// TwinCAT 3 PLC project ProyMain
// ProgramVersion: 3.1.4024.0
// libraries:
//   CmpBitmapPool, * (System)
//   Tc2_Standard, * (Beckhoff Automation GmbH)
//   Tc2_System, * (Beckhoff Automation GmbH)
//   Tc3_Module, * (Beckhoff Automation GmbH)
//   VisuDialogs, * (System)
// project tree:
//   DUTs/ E_GEMMA.TcDUT
//   / GlobalTextList.TcGTLO, PlcTask.TcTTO, Visualization Manager.TcVMO (not stored)
//   POUs/Estacion/ FB_Coordinador_SFC.TcPOU, FB_Director.TcPOU, FB_Estacion.TcPOU
//   POUs/ MAIN.TcPOU
//   POUs/Reloj/ FB_Clock.TcPOU
//   POUs/Tareas/ FB_AlimentadorVerificadorDesplazador_SFC.TcPOU, FB_CheckMaterial_SFC.TcPOU, FB_Descargador_SFC.TcPOU, FB_EstacionFinalizar_SFC.TcPOU, FB_EstacionPreparar_SFC.TcPOU, FB_Rechazador_SFC.TcPOU, FB_ResetDescargador_SFC.TcPOU, FB_SituarPale_SFC.TcPOU, FB_TransferirPale_SFC.TcPOU
//   VISUs/ ImagePool.TcIPO (not stored), Visualization.TcVIS
// real-time tasks:
//   TASK PlcTask: cycle T#10ms, priority 20, ADS port 350
// I/O:
//   DEVICE Device 1 (EtherCAT), AmsNetId 192.168.74.1.2.1
//     Term 1 (EK1200) [EK1200-5000 EtherCAT Power supply (2A E-Bus)]
//       Term 2 (EL1008) [EL1008 8Ch. Dig. Input 24V, 3ms]
//       Term 3 (EL1008) [EL1008 8Ch. Dig. Input 24V, 3ms]
//       Term 4 (EL2008) [EL2008 8Ch. Dig. Output 24V, 0.5A]
//       Term 5 (EL2008) [EL2008 8Ch. Dig. Output 24V, 0.5A]
//       Term 6 (EL1008) [EL1008 8Ch. Dig. Input 24V, 3ms]
//       Term 7 (EL1008) [EL1008 8Ch. Dig. Input 24V, 3ms]
//       Term 8 (EL2008) [EL2008 8Ch. Dig. Output 24V, 0.5A]
//       Term 9 (EL2008) [EL2008 8Ch. Dig. Output 24V, 0.5A]
//       Term 10 (EL9011) [EL9011 End Terminal]
//   DEVICE Device 2 (EtherCAT Automation Protocol), AmsNetId 192.168.74.1.3.1
//   DEVICE Device 3 (NOV-DP-RAM)
// variable links:
//   ProyMain/ProyMain Instance <-> Device 1 (EtherCAT)/Term 1 (EK1200)/Term 2 (EL1008)
//     PlcTask Inputs/MAIN.Estacion.Codigo_pale_bit_0 <-> Channel 7/Codigo de palé bit 0
//     PlcTask Inputs/MAIN.Estacion.Codigo_pale_bit_1 <-> Channel 8/Codigo de palé bit 1
//     PlcTask Inputs/MAIN.Estacion.EstacionConectada <-> Channel 5/Parte operativa conectada (armada)
//     PlcTask Inputs/MAIN.Estacion.Presencia_pale <-> Channel 6/presencia de palé
//     PlcTask Inputs/MAIN.Estacion.Pulsador_marcha <-> Channel 3/Pulsador de marcha
//     PlcTask Inputs/MAIN.Estacion.Pulsador_parada_NC <-> Channel 4/Pulsador de parada [NC]
//     PlcTask Inputs/MAIN.Estacion.Pulsador_parada_emergencia <-> Channel 1/Pulsador de parada de emergencia
//     PlcTask Inputs/MAIN.Estacion.Selector_modo_manual <-> Channel 2/Selector de modo manual
//   ProyMain/ProyMain Instance <-> Device 1 (EtherCAT)/Term 1 (EK1200)/Term 3 (EL1008)
//     PlcTask Inputs/MAIN.Estacion.Codigo_pale_bit_2 <-> Channel 1/Código de palé bit 2
//     PlcTask Inputs/MAIN.Estacion.Detector_presion <-> Channel 2/Detector de presión
//   ProyMain/ProyMain Instance <-> Device 1 (EtherCAT)/Term 1 (EK1200)/Term 4 (EL2008)
//     PlcTask Outputs/MAIN.Estacion.Activa_marcha_motor_cinta <-> Channel 5/Activa la marcha el motor de la cinta
//     PlcTask Outputs/MAIN.Estacion.Desconecta_parte_operativa <-> Channel 1/Desconecta parte operativa (desarma)
//     PlcTask Outputs/MAIN.Estacion.Invierte_marcha_motor_cinta <-> Channel 6/Invierte la marcha del motor de la cinta
//     PlcTask Outputs/MAIN.Estacion.Lampara_falta_material <-> Channel 4/Lámpara de falta material
//     PlcTask Outputs/MAIN.Estacion.Lampara_marcha <-> Channel 3/Lámpara de marcha
//     PlcTask Outputs/MAIN.Estacion.Retenedor_pale_baja <-> Channel 7/Cilindro del retenedor de palés baja
//     PlcTask Outputs/MAIN.Estacion.Separador_pale_sube <-> Channel 8/Cilindro del separador de palés sube
//   ProyMain/ProyMain Instance <-> Device 1 (EtherCAT)/Term 1 (EK1200)/Term 6 (EL1008)
//     PlcTask Inputs/MAIN.Estacion.Alimentador_detras <-> Channel 8/Cilindro del alimentador detrás
//     PlcTask Inputs/MAIN.Estacion.Desplazador_detras <-> Channel 7/Cilindro del desplazador detrás
//     PlcTask Inputs/MAIN.Estacion.Horizontal_descargador_delante <-> Channel 2/Cilindro horizontal del descargador delante (sobre el palé)
//     PlcTask Inputs/MAIN.Estacion.Horizontal_descargador_detras <-> Channel 1/Cilindro horizontal del descargador detrás (sobre el punto de descarga)
//     PlcTask Inputs/MAIN.Estacion.Verificador_abajo <-> Channel 6/Cilindro del verificador abajo
//     PlcTask Inputs/MAIN.Estacion.Verificador_arriba <-> Channel 5/Cilindro del verificador arriba
//     PlcTask Inputs/MAIN.Estacion.Vertical_descargador_abajo <-> Channel 4/Cilindro vertical del descargador abajo
//     PlcTask Inputs/MAIN.Estacion.Vertical_descargador_arriba <-> Channel 3/Cilindro vertical del descargador arriba
//   ProyMain/ProyMain Instance <-> Device 1 (EtherCAT)/Term 1 (EK1200)/Term 7 (EL1008)
//     PlcTask Inputs/MAIN.Estacion.Alimentador_delante <-> Channel 1/Cilindro del alimentador delante
//     PlcTask Inputs/MAIN.Estacion.Base_en_alimentador <-> Channel 3/Presencia de base en el alimentador
//     PlcTask Inputs/MAIN.Estacion.Vacio_obtenido_vacuostato_descargador <-> Channel 2/Vacío obtenido en el vacuostado del descargador
//   ProyMain/ProyMain Instance <-> Device 1 (EtherCAT)/Term 1 (EK1200)/Term 8 (EL2008)
//     PlcTask Outputs/MAIN.Estacion.Alimentador_adelante <-> Channel 7/Cilindro del alimentador adelante (hacia el punto de verificación)
//     PlcTask Outputs/MAIN.Estacion.Descargador_adelante <-> Channel 1/Cilindro del descargador adelante (hacia el palé)
//     PlcTask Outputs/MAIN.Estacion.Descargador_atras <-> Channel 2/Cilindro del descargador atrás (hacia el punto de descarga)
//     PlcTask Outputs/MAIN.Estacion.Descargador_baja <-> Channel 3/Cilindro del descargador baja
//     PlcTask Outputs/MAIN.Estacion.Desplazador_adelante <-> Channel 6/Cilindro del desplazador adelante (hacia el punto de descarga)
//     PlcTask Outputs/MAIN.Estacion.Eyector_succiona <-> Channel 8/Eyector de vacío del descargador succiona
//     PlcTask Outputs/MAIN.Estacion.Rechazador_adelante <-> Channel 4/Cilindro del rechazador adelante
//     PlcTask Outputs/MAIN.Estacion.Verificador_baja <-> Channel 5/Cilindro del verificador baja

CONFIGURATION ProyMain
    RESOURCE PLC ON TwinCAT3
        TASK PlcTask(INTERVAL := T#10ms, PRIORITY := 24);
        PROGRAM MAIN WITH PlcTask : MAIN;
    END_RESOURCE
END_CONFIGURATION

// ---- DUTs/E_GEMMA.TcDUT
{attribute 'qualified_only'}
{attribute 'strict'}
TYPE E_GEMMA :
(
    // Modos de la Guia de Estudio de los Modos de Marcha y Parada

    // Procedimientos de parada 
    A1, //  0: Parada en el estado inicial
    A2, //  1: Parada solicitada a final de ciclo 
    A3, //  2: Parada solicitada en un estado determinado
    A4, //  3: Parada obtenida
    A5, //  4: Preparacion para la recuperacion del fallo
    A6, //  5: Situando la PO en el estado inicial
    A7, //  6: Situando la PO en un estado determinado

    // Procedimientos de funcionamiento
    F1, //  7: Produccion normal
    F2, //  8: Secuencia de preparacion
    F3, //  9: Secuencia de finalizacion
    F4, // 10: Verificacion en desorden
    F5, // 11: Verificacion en orden
    F6, // 12: Secuencia de prueba

    // Procedimientos de fallo
    D1, // 13: Parada de emergencia
    D2, // 14: Diagnostico y/o tratamiento de los fallos
    D3  // 15: Produccion a pesar de los fallos
);
END_TYPE

// ---- POUs/MAIN.TcPOU
PROGRAM MAIN
VAR
    Estacion: FB_Estacion;
END_VAR

Estacion();

END_PROGRAM

// ---- POUs/Estacion/FB_Estacion.TcPOU
FUNCTION_BLOCK FB_Estacion
VAR_INPUT
    EstadoPausa: BOOL;
    EstadoReinicia: BOOL;
    CiclosSolicitados: UINT := 0;
    
    Tcheck: TIME := T#1S;
    Treset: TIME := T#1S;
    Tdesplazador: TIME := T#1S;
	Tcinta: TIME := T#0.5S;
END_VAR
VAR_OUTPUT
    CondicionInicial: BOOL := TRUE;
    CiclosPendientes: UINT;
    CiclosAceptados: UINT;
	CiclosRechazados: UINT;
    PaleCodigo: BYTE;
	pieza_ok: BOOL;
    
    // Entradas comunes
	Base_en_alimentador AT %I*: BOOL;
    Pulsador_parada_emergencia AT %I*: BOOL;
    Selector_modo_manual AT %I*: BOOL;
    Pulsador_marcha AT %I*: BOOL;
    Pulsador_parada_NC AT %I*: BOOL := TRUE; // Contacto normalmente cerrado
    EstacionConectada AT %I*: BOOL := TRUE;
    Detector_presion AT %I*: BOOL := TRUE;

    Presencia_pale AT %I*: BOOL;
    Codigo_pale_bit_0 AT %I*: BOOL;
    Codigo_pale_bit_1 AT %I*: BOOL;
    Codigo_pale_bit_2 AT %I*: BOOL;

    // Entradas espeficicas
    //Terminal 6
	Horizontal_descargador_detras AT %I*: BOOL;
	Horizontal_descargador_delante AT %I*: BOOL;
	Vertical_descargador_arriba AT %I*: BOOL;
	Vertical_descargador_abajo AT %I*: BOOL;
	Verificador_arriba AT %I*: BOOL;
	Verificador_abajo AT %I*: BOOL;
	Desplazador_detras AT %I*: BOOL;
	Desplazador_delante AT %I*: BOOL;
	Alimentador_detras AT %I*: BOOL;
	
	
	//Terminal 7
	Alimentador_delante AT %I*: BOOL;
	Vacio_obtenido_vacuostato_descargador AT %I*: BOOL;

END_VAR
VAR
	ModoAnterior: E_GEMMA;    

    // Bloques funcionales
    CLK: FB_Clock;	

    // Bloques funcionales
	Director : FB_Director;
    Coordinador: FB_Coordinador_SFC;
	ChequeaMaterial: FB_CheckMaterial_SFC;
	AlimentadorVerificadorDesplazador: FB_AlimentadorVerificadorDesplazador_SFC;
    SituarPale: FB_SituarPale_SFC;
	ResetDescargador: FB_ResetDescargador_SFC;
    Descargador: FB_Descargador_SFC;
    Rechazador: FB_Rechazador_SFC;
    TransferirPale: FB_TransferirPale_SFC;
	Finalizar: FB_EstacionFinalizar_SFC;
	Preparar: FB_EstacionPreparar_SFC;
    
    // Salidas comunes
    Desconecta_parte_operativa AT %Q*: BOOL;
    Lampara_falta_material AT %Q*: BOOL;
    Lampara_marcha AT %Q*: BOOL;
    Lampara_alarma AT %Q*: BOOL;

    Activa_marcha_motor_cinta AT %Q*: BOOL;
    Invierte_marcha_motor_cinta AT %Q*: BOOL;
    Retenedor_pale_baja AT %Q*: BOOL;
    Separador_pale_sube AT %Q*: BOOL;
    
    //Terminal 8
	Descargador_adelante AT %Q*: BOOL;
	Descargador_atras AT %Q*: BOOL;
	Descargador_baja AT %Q*: BOOL;
	Rechazador_adelante AT %Q*: BOOL;
	Verificador_baja AT %Q*: BOOL;
	Desplazador_adelante AT %Q*: BOOL;
	Alimentador_adelante AT %Q*: BOOL;
	Eyector_succiona AT %Q*: BOOL;
	SFCPause: BOOL;
END_VAR

// Modo Automático
//IF NOT Selector_Modo_Manual THEN
CLK();

    // Bloques Funcionales
    Director(
        CondicionInicial := CondicionInicial,
        CondicionMarcha:= (CiclosSolicitados > 0) AND CondicionInicial,
        Emergencia := Pulsador_parada_emergencia,
        Finalizada := Finalizar.Done,
        FinTarea := (CiclosPendientes = 0),
        FinCiclo := Coordinador.Done,
        Manual := Selector_modo_manual,
        Marcha := Pulsador_marcha,
        ParaCiclo := NOT Pulsador_parada_NC,
        Preparada := Preparar.Done,
        Reinicia := EstadoReinicia
    );
	
	IF (Director.Modo <> E_GEMMA.F4) THEN

    SituarPale( //SituarPale
        SFCPause := NOT EstadoReinicia AND EstadoPausa,
        SFCReset := EstadoReinicia,
        Ack := NOT Coordinador.SituaPale,
        Execute := Coordinador.SituaPale,
        Tcinta := Tcinta,
        Presencia_pale := Presencia_pale,
           //Codigo_pale_bit_0 := Codigo_pale_bit_0,
        //Codigo_pale_bit_1 := Codigo_pale_bit_1,
        //Codigo_pale_bit_2 := Codigo_pale_bit_2

    );

	// Bloques Funcionales
	Coordinador(

		CiclosPendientes := CiclosPendientes,
		CiclosAceptados := CiclosAceptados,
		CiclosSolicitados := CiclosSolicitados,
		CiclosRechazados := CiclosRechazados,
		SFCPause := NOT EstadoReinicia AND EstadoPausa,
        SFCReset := EstadoReinicia,
		Ack := TRUE,
        Execute := (Director.Modo = E_GEMMA.F1),
		PaleSituado := SituarPale.Done,
		HayMaterial := ChequeaMaterial.Done,
		Verificado := AlimentadorVerificadorDesplazador.Done,
		DescargadorReseteado := ResetDescargador.Done,
        Rechazado := Rechazador.Done,
		BaseCargada := Descargador.Done,
		PaleTransferido := TransferirPale.Done,
		pieza_ok := pieza_ok
		
	);
	
	Preparar(
		
		SFCPause := NOT EstadoReinicia AND EstadoPausa,
        SFCReset := EstadoReinicia,
        Ack := (Director.Modo <> E_GEMMA.F2),
        Execute := (Director.Modo = E_GEMMA.F2),
		Horizontal_descargador_detras := Horizontal_descargador_detras,
		Vertical_descargador_arriba := Vertical_descargador_arriba,
		Presencia_pale := Presencia_pale
	
	);
	
	Finalizar(
		
		SFCPause := NOT EstadoReinicia AND EstadoPausa,
        SFCReset := EstadoReinicia,
        Ack := (Director.Modo <> E_GEMMA.F3),
        Execute := (Director.Modo = E_GEMMA.F3),
		Horizontal_descargador_detras := Horizontal_descargador_detras,
		Vertical_descargador_arriba := Vertical_descargador_arriba,
		Presencia_pale := Presencia_pale
	
	);
	
	SituarPale(

		SFCPause := NOT EstadoReinicia AND EstadoPausa,
        SFCReset := EstadoReinicia,
        Ack := NOT Coordinador.SituaPale,
        Execute := Coordinador.SituaPale,
        Tcinta := Tcinta,
        Presencia_pale := Presencia_pale,
       	//Codigo_pale_bit_0 := Codigo_pale_bit_0,
        //Codigo_pale_bit_1 := Codigo_pale_bit_1,
        //Codigo_pale_bit_2 := Codigo_pale_bit_2

	);
	
	ChequeaMaterial(
		Ack := NOT Coordinador.ChequeaMaterial,
		SFCPause := NOT EstadoReinicia AND EstadoPausa,
        SFCReset := EstadoReinicia,
		Execute := Coordinador.ChequeaMaterial,
		Base_en_Alimentador := Base_en_alimentador,
		Pulsador_marcha := Pulsador_marcha
	);
	
	AlimentadorVerificadorDesplazador(
		
		Ack := NOT Coordinador.VerificaBase,
        Tcheck := Tcheck,
		SFCPause := NOT EstadoReinicia AND EstadoPausa,
        SFCReset := EstadoReinicia,
		Execute := Coordinador.VerificaBase,
		Alimentador_delante := Alimentador_delante,
		Alimentador_detras := Alimentador_detras,
		Verificador_arriba := Verificador_arriba ,
		Verificador_abajo := Verificador_abajo,
		Desplazador_delante := Desplazador_delante,
		Desplazador_detras := Desplazador_detras, 
		
	);
	
	ResetDescargador(

		Ack := NOT Coordinador.ResetDescargador,
		SFCPause := NOT EstadoReinicia AND EstadoPausa,
        SFCReset := EstadoReinicia,
		Execute := Coordinador.ResetDescargador,
		Horizontal_descargador_detras := Horizontal_descargador_detras,
		Vertical_descargador_arriba := Vertical_descargador_arriba
	);
	
	Descargador(
		
		Ack := NOT Coordinador.CargaBase,
		SFCPause := NOT EstadoReinicia AND EstadoPausa,
        SFCReset := EstadoReinicia,
		Execute := Coordinador.CargaBase,
		Horizontal_descargador_detras := Horizontal_descargador_detras,
		Vertical_descargador_abajo := Vertical_descargador_abajo,
		Vacio_obtenido_vacuostato_descargador := Vacio_obtenido_vacuostato_descargador ,
		Vertical_descargador_arriba := Vertical_descargador_arriba ,
		Horizontal_descargador_delante := Horizontal_descargador_delante ,
	
	);	
		
	Rechazador(
		
		Ack := NOT Coordinador.RechazaBase,
		SFCPause := NOT EstadoReinicia AND EstadoPausa,
        SFCReset := EstadoReinicia,
		Execute := Coordinador.RechazaBase,
		Verificador_abajo := Verificador_abajo
		
	);
	
	TransferirPale(
	
		Ack := NOT Coordinador.TransfierePale,
		SFCPause := NOT EstadoReinicia AND EstadoPausa,
        SFCReset := EstadoReinicia,
		Execute := Coordinador.TransfierePale,
		Presencia_pale:=Presencia_pale

	);
	
	//Acciones Comunes
	// Parametros de Salida
	//Lampara_falta_material := ChequeaMaterial.Lampara_falta_material;
	Activa_marcha_motor_cinta := SituarPale.Activa_marcha_motor_cinta OR TransferirPale.Activa_marcha_motor_cinta OR Preparar.Activa_marcha_motor_cinta OR Finalizar.Activa_marcha_motor_cinta;
	//CheckMaterial
	Lampara_alarma := ChequeaMaterial.LamparaAlarma;
	Lampara_falta_material := ChequeaMaterial.Lampara_falta_material;
	//TranferirPale
	 Retenedor_pale_baja := TransferirPale.Retenedor_pale_baja;
	 Separador_pale_sube := TransferirPale.Separador_pale_sube;
	//AlimentadorVerificadorDesplazador
	Alimentador_adelante := AlimentadorVerificadorDesplazador.Alimentador_adelante;
	Verificador_baja := AlimentadorVerificadorDesplazador.Verificador_baja;
	Desplazador_adelante := AlimentadorVerificadorDesplazador.Desplazador_adelante;
	pieza_ok := AlimentadorVerificadorDesplazador.pieza_ok;
	//Descargador
	Eyector_succiona := Descargador.Eyector_succiona;
	Descargador_adelante := Descargador.Descargador_adelante;
	Descargador_atras := Descargador.Descargador_atras OR ResetDescargador.Descargador_atras;
	Descargador_baja := Descargador.Descargador_baja;
	//Rechazador
	Rechazador_adelante := Rechazador.Rechazador_adelante;
	
	IF NOT EstadoPausa THEN
	
		EstadoPausa := not Pulsador_parada_NC;
	
	ELSE
	
		EstadoPausa := NOT Pulsador_marcha;
	
	END_IF

END_IF	
	
// Parametros de Salida
CondicionInicial := EstacionConectada; //AND Desplazador_detras AND Verificador_arriba AND Vertical_descargador_arriba AND Alimentador_detras;

//al iniciar una tarea
IF ((ModoAnterior = E_GEMMA.A1) AND (Director.Modo <> E_GEMMA.A1) AND (CiclosPendientes = 0)) THEN
    CiclosPendientes := CiclosSolicitados;
END_IF

//IF (Director.Modo <> E_GEMMA.F4) THEN
    //PaleCodigo := SituarPale.PaleCodigo;
//ELSE 
    //PaleCodigo.0 := Codigo_pale_bit_0;
    //PaleCodigo.1 := Codigo_pale_bit_1;
    //PaleCodigo.2 := Codigo_pale_bit_2;
//END_IF

// ACTULIZACION DE IMAGENES
ModoAnterior := Director.Modo;

END_FUNCTION_BLOCK

// ---- POUs/Reloj/FB_Clock.TcPOU
FUNCTION_BLOCK FB_Clock
(*
Square wave oscillator

Copyright (c) 2009-2017 victortorreslopez

GNU General Public License

Version history
2.1, 2017/03/15, VTL: style review (PLCopen Coding Guidelines)
2.0, 2014/12/29, VTL: complete review
1.0, 2009/11/06, VTL: first release
0.0, 2009/11/06, VTL: alfa release
*)
VAR_INPUT
  EN: BOOL := TRUE;	(* ENabled *)
  PT: TIME := T#500ms; (* Semicycle time *)
END_VAR
VAR_OUTPUT
  ET: TIME; (* Elapsed time *)
  Q: BOOL; (* Square wave *)
END_VAR
VAR
  Timer: TON; (* Auto-pilot timer *)
END_VAR

(* OUTPUT FUNCTION *)
IF Timer.Q THEN
  Q := NOT Q;
END_IF

(* FUNCTION BLOCKS *)
Timer(IN := EN AND NOT Timer.Q, PT := PT, ET => ET);

END_FUNCTION_BLOCK

// ---- POUs/Estacion/FB_Director.TcPOU
FUNCTION_BLOCK FB_Director
VAR_INPUT
    CondicionInicial: BOOL; // Condiciones materiales necesarias para iniciar la produccion
    CondicionMarcha: BOOL; // Condiciones logicas necesarias para iniciar la produccion
    Emergencia: BOOL;
    Finalizada: BOOL;
    FinTarea: BOOL;
    FinCiclo: BOOL;
    Manual: BOOL;
    Marcha: BOOL;
    ParaCiclo: BOOL;
    Preparada: BOOL;
    Reinicia: BOOL;
END_VAR
VAR_OUTPUT
    Modo: E_GEMMA := E_GEMMA.A6;

    Defecto: BOOL; // Procedimientos de defecto
    Funcionamiento: BOOL; // Procedimientos de funcionamiento
    Parada: BOOL; // Procedimientos de parada
    Produccion: BOOL; // Procedimientos que proporcionan valor añadido
END_VAR

// FUNCION DE ESTADO
IF Emergencia THEN
    Modo := E_GEMMA.D1;
ELSIF Reinicia THEN
    Modo := E_GEMMA.A6;
ELSE
    CASE Modo OF
        // Procedimientos de parada
        E_GEMMA.A1: // Parada en el estado inicial
            IF NOT CondicionInicial THEN
                Modo := E_GEMMA.A6;
            ELSIF Manual THEN
                Modo := E_GEMMA.F4;
            ELSIF (CondicionMarcha AND Marcha) THEN
                Modo := E_GEMMA.F2;
            END_IF
        E_GEMMA.A2: // Parada solicitada a final de ciclo
            IF FinCiclo THEN
                Modo := E_GEMMA.A1;
            END_IF
        E_GEMMA.A3: // Parada solicitada en un estado determinado 
            ;
        E_GEMMA.A4: // Parada obtenida 
            ;
        E_GEMMA.A5: // Preparando de reanudacion tras el fallo 
            ;
        E_GEMMA.A6: // Situando la PO en el estado inicial 
            IF CondicionInicial THEN
                Modo := E_GEMMA.A1;
            ELSIF Manual THEN
                Modo := E_GEMMA.F4;
            END_IF
        E_GEMMA.A7: // Situando la PO en un estado determinado 
            ;

        // Procedimientos de funcionamiento 
        E_GEMMA.F1: // Produccion normal 
            IF FinTarea THEN
                Modo := E_GEMMA.F3;
            ELSIF ParaCiclo THEN
                Modo := E_GEMMA.A2;
            END_IF
        E_GEMMA.F2: // Secuencia de preparacion 
            IF Preparada THEN
                Modo := E_GEMMA.F1;
            END_IF
        E_GEMMA.F3: // Secuencia de finalizacion 
            IF Finalizada THEN
                Modo := E_GEMMA.A1;
            END_IF
        E_GEMMA.F4: // Verificacion sin orden 
            IF NOT Manual THEN
                Modo := E_GEMMA.A6;
            END_IF
        E_GEMMA.F5: // Verificacion en orden 
            ;
        E_GEMMA.F6: // Prueba 
            ;

        // Procedimientos de defecto 
        E_GEMMA.D1: // Parada de emergencia 
            IF NOT Emergencia THEN
                Modo := E_GEMMA.A6;
            END_IF
        E_GEMMA.D2: // Diagnostico/tratamiento de los fallos 
            ;
        E_GEMMA.D3: // Produccion a pesar de los fallos 
            ;
    END_CASE
END_IF

// PARAMETROS DE SALIDA 
Defecto := (Modo >= E_GEMMA.D1) AND (Modo <= E_GEMMA.D3);
Funcionamiento:= (Modo >= E_GEMMA.F1) AND (Modo <= E_GEMMA.F6);
Parada := (Modo >= E_GEMMA.A1) AND (Modo <= E_GEMMA.A7);
Produccion := (Modo = E_GEMMA.A2) OR (Modo = E_GEMMA.A3) OR (Modo = E_GEMMA.F1) 
    OR (Modo = E_GEMMA.F2) OR (Modo = E_GEMMA.F3) OR (Modo = E_GEMMA.F5)
    OR (Modo = E_GEMMA.F6) OR (Modo = E_GEMMA.D3);

END_FUNCTION_BLOCK

// ---- POUs/Estacion/FB_Coordinador_SFC.TcPOU
FUNCTION_BLOCK FB_Coordinador_SFC

VAR_IN_OUT
	CiclosPendientes: UINT;
	CiclosAceptados: UINT;
	CiclosRechazados: UINT;
END_VAR
VAR_INPUT
	// SFC-Flags
    SFCPause: BOOL;
    SFCReset: BOOL;
    
    // Indicadores de sincronizacion
    Ack: BOOL := TRUE; //evita que la tarea se realice dos veces
    Execute: BOOL; 
    
    // Parametros de sincronizacion
    PaleSituado: BOOL;
	HayMaterial: BOOL;
    Verificado: BOOL;
	Rechazado: BOOL;
	DescargadorReseteado: BOOL;
    BaseCargada: BOOL;
    PaleTransferido: BOOL;
    
    // Parametros
    CondicionInicial: BOOL;
    CiclosSolicitados: UINT;
	
	//Entradas
	Base_en_Alimentador: BOOL;
	pieza_ok: BOOL;
END_VAR
VAR_OUTPUT
	// Indicadores de sincronizacion
    Done: BOOL;
    Ready: BOOL;

    // Parametros de sincronizacion
    SituaPale: BOOL;
	ChequeaMaterial: BOOL;
    VerificaBase: BOOL;
	ResetDescargador: BOOL;
    RechazaBase: BOOL;
	CargaBase: BOOL;
    TransfierePale: BOOL;
    
    // Salidas
    LamparaAlarma: BOOL;
    LamparaMarcha: BOOL;
	Lampara_falta_material: BOOL;
END_VAR
VAR
	// Bloques funcionales
    CLK: FB_Clock;
END_VAR

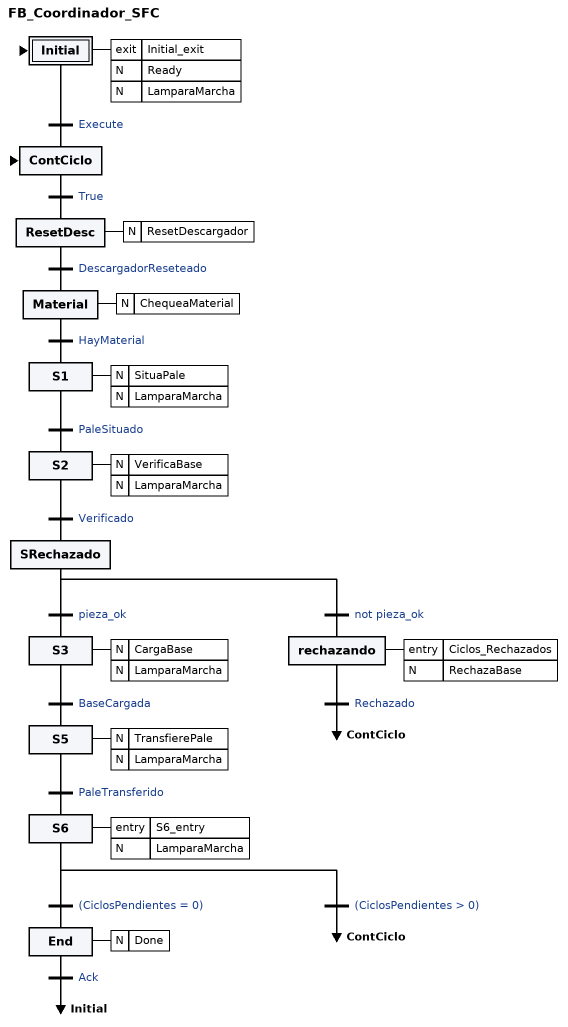
INITIAL_STEP Initial:
    Initial_exit(P0);  // exit action
    Ready(N);
    LamparaMarcha(N);
END_STEP
TRANSITION FROM Initial TO ContCiclo
    := Execute;
END_TRANSITION
STEP ContCiclo:
END_STEP
TRANSITION FROM ContCiclo TO ResetDesc
    := True;
END_TRANSITION
STEP ResetDesc:
    ResetDescargador(N);
END_STEP
TRANSITION FROM ResetDesc TO Material
    := DescargadorReseteado;
END_TRANSITION
STEP Material:
    ChequeaMaterial(N);
END_STEP
TRANSITION FROM Material TO S1
    := HayMaterial;
END_TRANSITION
STEP S1:
    SituaPale(N);
    LamparaMarcha(N);
END_STEP
TRANSITION FROM S1 TO S2
    := PaleSituado;
END_TRANSITION
STEP S2:
    VerificaBase(N);
    LamparaMarcha(N);
END_STEP
TRANSITION FROM S2 TO SRechazado
    := Verificado;
END_TRANSITION
STEP SRechazado:
END_STEP
TRANSITION FROM SRechazado TO S3
    := pieza_ok;
END_TRANSITION
TRANSITION FROM SRechazado TO rechazando
    := not pieza_ok;
END_TRANSITION
STEP rechazando:
    Ciclos_Rechazados(P1);  // entry action
    RechazaBase(N);
END_STEP
TRANSITION FROM rechazando TO ContCiclo
    := Rechazado;
END_TRANSITION
STEP S3:
    CargaBase(N);
    LamparaMarcha(N);
END_STEP
TRANSITION FROM S3 TO S5
    := BaseCargada;
END_TRANSITION
STEP S5:
    TransfierePale(N);
    LamparaMarcha(N);
END_STEP
TRANSITION FROM S5 TO S6
    := PaleTransferido;
END_TRANSITION
STEP S6:
    S6_entry(P1);  // entry action
    LamparaMarcha(N);
END_STEP
TRANSITION FROM S6 TO End
    := (CiclosPendientes = 0);
END_TRANSITION
TRANSITION FROM S6 TO ContCiclo
    := (CiclosPendientes > 0);
END_TRANSITION
STEP End:
    Done(N);
END_STEP
TRANSITION FROM End TO Initial
    := Ack;
END_TRANSITION

ACTION Ciclos_Rechazados:
CiclosRechazados := CiclosRechazados + 1;
END_ACTION

ACTION Initial_exit:
IF (CiclosPendientes = 0) THEN
	CiclosPendientes := CiclosSolicitados;
	CiclosRechazados := 0;
	CiclosAceptados := 0;
END_IF
END_ACTION

ACTION S6_entry:
CiclosPendientes := CiclosPendientes - 1;
CiclosAceptados := CiclosAceptados + 1;
END_ACTION

END_FUNCTION_BLOCK

// ---- POUs/Tareas/FB_CheckMaterial_SFC.TcPOU
FUNCTION_BLOCK FB_CheckMaterial_SFC
VAR_INPUT
	// SFC-Flags
    SFCPause: BOOL;
    SFCReset: BOOL;
    
    // Indicadores de sincronizacion
    Ack: BOOL := TRUE; 
    Execute: BOOL;
	
	//Entradas
	Base_en_Alimentador: BOOL;
	Pulsador_marcha: BOOL;
END_VAR
VAR_OUTPUT
	// Indicadores de sincronizacion
    Done: BOOL;
    Ready: BOOL;
	
	//Salidas
	LamparaAlarma: BOOL;
	Lampara_falta_material: BOOL;
END_VAR
VAR
	TMAt: TIME := T#1S;
END_VAR

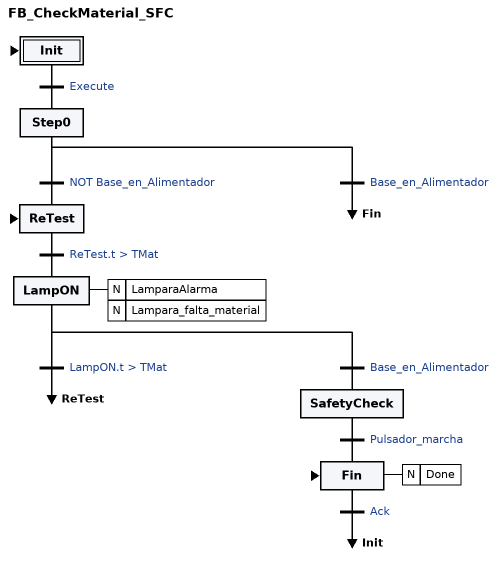
INITIAL_STEP Init:
END_STEP
TRANSITION FROM Init TO Step0
    := Execute;
END_TRANSITION
STEP Step0:
END_STEP
TRANSITION FROM Step0 TO ReTest
    := NOT Base_en_Alimentador;
END_TRANSITION
STEP ReTest:
END_STEP
TRANSITION FROM ReTest TO LampON
    := ReTest.t > TMat;
END_TRANSITION
TRANSITION FROM Step0 TO Fin
    := Base_en_Alimentador;
END_TRANSITION
STEP LampON:
    LamparaAlarma(N);
    Lampara_falta_material(N);
END_STEP
TRANSITION FROM LampON TO ReTest
    := LampON.t > TMat;
END_TRANSITION
TRANSITION FROM LampON TO SafetyCheck
    := Base_en_Alimentador;
END_TRANSITION
STEP SafetyCheck:
END_STEP
TRANSITION FROM SafetyCheck TO Fin
    := Pulsador_marcha;
END_TRANSITION
STEP Fin:
    Done(N);
END_STEP
TRANSITION FROM Fin TO Init
    := Ack;
END_TRANSITION

END_FUNCTION_BLOCK

// ---- POUs/Tareas/FB_AlimentadorVerificadorDesplazador_SFC.TcPOU
FUNCTION_BLOCK FB_AlimentadorVerificadorDesplazador_SFC
VAR_INPUT
	//Tiempo
	Tcheck: TIME := T#1S;
	Tdesplazador: TIME := T#1S;
	
	// SFC-Flags
	SFCPause: BOOL;
	SFCReset: BOOL;
	
	//Indicadores de sincronizacion
	Ack: BOOL:= TRUE;
	Execute: BOOL;
	
	//Entradas
	
	Alimentador_delante: BOOL; //Bajo el verificador
	Alimentador_detras: BOOL;
	Verificador_arriba: BOOL;
	Verificador_abajo: BOOL;
	Desplazador_delante: BOOL;
	Desplazador_detras: BOOL;
	
END_VAR
VAR_OUTPUT
	//indicadores de sincronizacion
	Done: BOOL;
	Ready: BOOL;

	//Salidas
	Alimentador_adelante: BOOL;
	Verificador_baja: BOOL;
	Desplazador_adelante: BOOL;
	
	pieza_ok : BOOL;

END_VAR
VAR
END_VAR

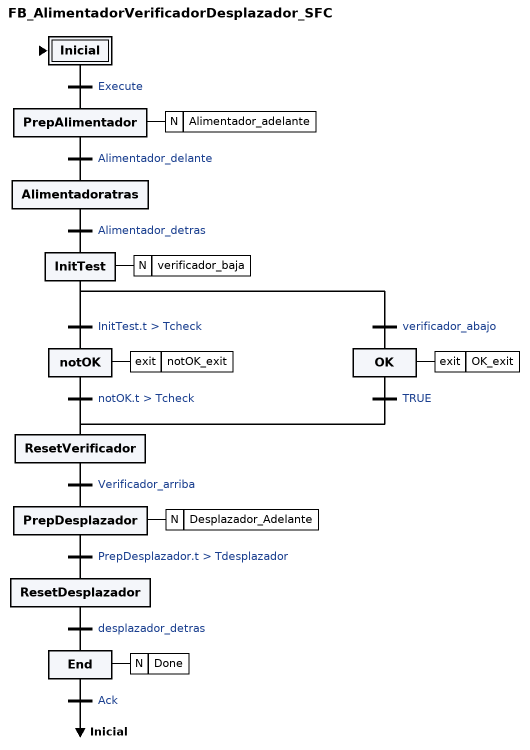
INITIAL_STEP Inicial:
END_STEP
TRANSITION FROM Inicial TO PrepAlimentador
    := Execute;
END_TRANSITION
STEP PrepAlimentador:
    Alimentador_adelante(N);
END_STEP
TRANSITION FROM PrepAlimentador TO Alimentadoratras
    := Alimentador_delante;
END_TRANSITION
STEP Alimentadoratras:
END_STEP
TRANSITION FROM Alimentadoratras TO InitTest
    := Alimentador_detras;
END_TRANSITION
STEP InitTest:
    verificador_baja(N);
END_STEP
TRANSITION FROM InitTest TO notOK
    := InitTest.t > Tcheck;
END_TRANSITION
STEP notOK:
    notOK_exit(P0);  // exit action
END_STEP
TRANSITION FROM notOK TO ResetVerificador
    := notOK.t > Tcheck;
END_TRANSITION
TRANSITION FROM InitTest TO OK
    := verificador_abajo;
END_TRANSITION
STEP OK:
    OK_exit(P0);  // exit action
END_STEP
TRANSITION FROM OK TO ResetVerificador
    := TRUE;
END_TRANSITION
STEP ResetVerificador:
END_STEP
TRANSITION FROM ResetVerificador TO PrepDesplazador
    := Verificador_arriba;
END_TRANSITION
STEP PrepDesplazador:
    Desplazador_Adelante(N);
END_STEP
TRANSITION FROM PrepDesplazador TO ResetDesplazador
    := PrepDesplazador.t > Tdesplazador;
END_TRANSITION
STEP ResetDesplazador:
END_STEP
TRANSITION FROM ResetDesplazador TO End
    := desplazador_detras;
END_TRANSITION
STEP End:
    Done(N);
END_STEP
TRANSITION FROM End TO Inicial
    := Ack;
END_TRANSITION

ACTION notOK_exit:
pieza_ok := FALSE;
END_ACTION

ACTION OK_exit:
pieza_ok := TRUE;
END_ACTION

END_FUNCTION_BLOCK

// ---- POUs/Tareas/FB_SituarPale_SFC.TcPOU
FUNCTION_BLOCK FB_SituarPale_SFC
VAR_INPUT
	//nuestras_variables
	Tcinta: TIME := T#0.5S;

	
    // SFC-Flags
    SFCPause: BOOL;
    SFCReset: BOOL;
    
    // Indicadores de sincronizacion
    Ack: BOOL := TRUE;
    Execute: BOOL;
	
	//Entradas
   	Presencia_pale: BOOL;
	Vertical_descargador_abajo: BOOL;
	Vacio_obtenido_vacuostato_descargador: BOOL;
	Vertical_descargador_arriba: BOOL;
	Horizontal_descargador_delante: BOOL;
	
	
	
END_VAR
VAR_OUTPUT
    // Indicadores de sincronizacion
    Done: BOOL;
    Ready: BOOL;

	//Salidas
	Activa_marcha_motor_cinta: BOOL;
END_VAR
VAR
END_VAR

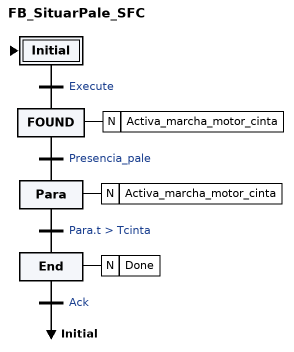
INITIAL_STEP Initial:
END_STEP
TRANSITION FROM Initial TO FOUND
    := Execute;
END_TRANSITION
STEP FOUND:
    Activa_marcha_motor_cinta(N);
END_STEP
TRANSITION FROM FOUND TO Para
    := Presencia_pale;
END_TRANSITION
STEP Para:
    Activa_marcha_motor_cinta(N);
END_STEP
TRANSITION FROM Para TO End
    := Para.t > Tcinta;
END_TRANSITION
STEP End:
    Done(N);
END_STEP
TRANSITION FROM End TO Initial
    := Ack;
END_TRANSITION

END_FUNCTION_BLOCK

// ---- POUs/Tareas/FB_ResetDescargador_SFC.TcPOU
FUNCTION_BLOCK FB_ResetDescargador_SFC

VAR_INPUT
	//nuestras_variables

    // SFC-Flags
    SFCPause: BOOL;
    SFCReset: BOOL;
    
    // Indicadores de sincronizacion
    Ack: BOOL := TRUE;
    Execute: BOOL;
	
	//Entradas
    Horizontal_descargador_detras: BOOL;
	Vertical_descargador_arriba: BOOL;

	
END_VAR
VAR_OUTPUT
    // Indicadores de sincronizacion
    Done: BOOL;
    Ready: BOOL;

	//Salidas
	Descargador_atras: BOOL;
	
END_VAR
VAR
END_VAR

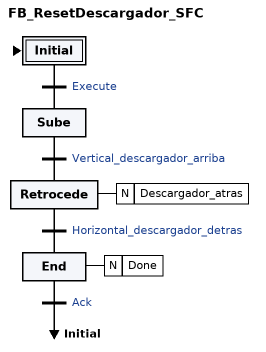
INITIAL_STEP Initial:
END_STEP
TRANSITION FROM Initial TO Sube
    := Execute;
END_TRANSITION
STEP Sube:
END_STEP
TRANSITION FROM Sube TO Retrocede
    := Vertical_descargador_arriba;
END_TRANSITION
STEP Retrocede:
    Descargador_atras(N);
END_STEP
TRANSITION FROM Retrocede TO End
    := Horizontal_descargador_detras;
END_TRANSITION
STEP End:
    Done(N);
END_STEP
TRANSITION FROM End TO Initial
    := Ack;
END_TRANSITION

END_FUNCTION_BLOCK

// ---- POUs/Tareas/FB_Descargador_SFC.TcPOU
FUNCTION_BLOCK FB_Descargador_SFC
VAR_INPUT
	//nuestras_variables
	pieza_ok: BOOL;	

    // SFC-Flags
    SFCPause: BOOL;
    SFCReset: BOOL;
    
    // Indicadores de sincronizacion
    Ack: BOOL := TRUE;
    Execute: BOOL;
	
	//Entradas
    Horizontal_descargador_detras: BOOL;
	Vertical_descargador_abajo: BOOL;
	Vacio_obtenido_vacuostato_descargador: BOOL;
	Vertical_descargador_arriba: BOOL;
	Horizontal_descargador_delante: BOOL;

	
END_VAR
VAR_OUTPUT
    // Indicadores de sincronizacion
    Done: BOOL;
    Ready: BOOL;

	//Salidas
	Descargador_atras: BOOL;
	Descargador_baja: BOOL;
	Eyector_succiona: BOOL;
	Descargador_adelante: BOOL;
END_VAR
VAR
END_VAR

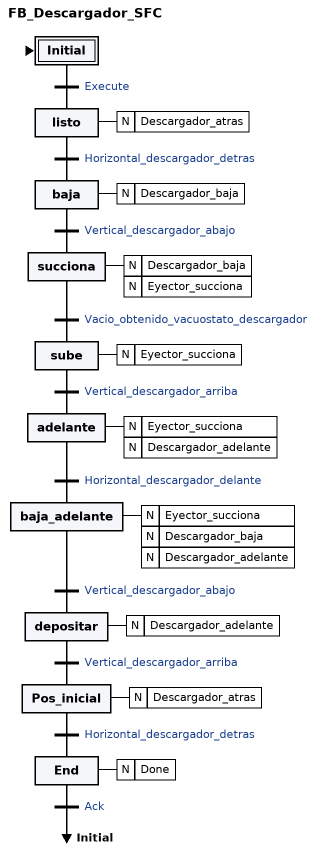
INITIAL_STEP Initial:
END_STEP
TRANSITION FROM Initial TO listo
    := Execute;
END_TRANSITION
STEP listo:
    Descargador_atras(N);
END_STEP
TRANSITION FROM listo TO baja
    := Horizontal_descargador_detras;
END_TRANSITION
STEP baja:
    Descargador_baja(N);
END_STEP
TRANSITION FROM baja TO succiona
    := Vertical_descargador_abajo;
END_TRANSITION
STEP succiona:
    Descargador_baja(N);
    Eyector_succiona(N);
END_STEP
TRANSITION FROM succiona TO sube
    := Vacio_obtenido_vacuostato_descargador;
END_TRANSITION
STEP sube:
    Eyector_succiona(N);
END_STEP
TRANSITION FROM sube TO adelante
    := Vertical_descargador_arriba;
END_TRANSITION
STEP adelante:
    Eyector_succiona(N);
    Descargador_adelante(N);
END_STEP
TRANSITION FROM adelante TO baja_adelante
    := Horizontal_descargador_delante;
END_TRANSITION
STEP baja_adelante:
    Eyector_succiona(N);
    Descargador_baja(N);
    Descargador_adelante(N);
END_STEP
TRANSITION FROM baja_adelante TO depositar
    := Vertical_descargador_abajo;
END_TRANSITION
STEP depositar:
    Descargador_adelante(N);
END_STEP
TRANSITION FROM depositar TO Pos_inicial
    := Vertical_descargador_arriba;
END_TRANSITION
STEP Pos_inicial:
    Descargador_atras(N);
END_STEP
TRANSITION FROM Pos_inicial TO End
    := Horizontal_descargador_detras;
END_TRANSITION
STEP End:
    Done(N);
END_STEP
TRANSITION FROM End TO Initial
    := Ack;
END_TRANSITION

END_FUNCTION_BLOCK

// ---- POUs/Tareas/FB_Rechazador_SFC.TcPOU
FUNCTION_BLOCK FB_Rechazador_SFC
VAR_INPUT
	
	//Tiempo
	Tcheck: TIME := T#1S;	
	
	// SFC-Flags
	SFCPause: BOOL;
	SFCReset: BOOL;
	
	//Indicadores de sincronizacion
	Ack: BOOL:= TRUE;
	Execute: BOOL;
	
	//Entradas
	
	Verificador_abajo: BOOL;

	
END_VAR
VAR_OUTPUT
	//indicadores de sincronizacion
	Done: BOOL;
	Ready: BOOL;

	//Salidas
	Rechazador_adelante: BOOL;
	
END_VAR
VAR
END_VAR

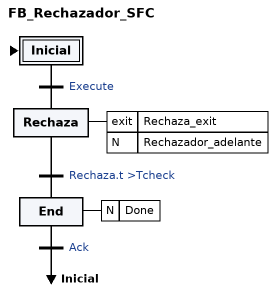
INITIAL_STEP Inicial:
END_STEP
TRANSITION FROM Inicial TO Rechaza
    := Execute;
END_TRANSITION
STEP Rechaza:
    Rechaza_exit(P0);  // exit action
    Rechazador_adelante(N);
END_STEP
TRANSITION FROM Rechaza TO End
    := Rechaza.t >Tcheck;
END_TRANSITION
STEP End:
    Done(N);
END_STEP
TRANSITION FROM End TO Inicial
    := Ack;
END_TRANSITION

ACTION Rechaza_exit:

END_ACTION

END_FUNCTION_BLOCK

// ---- POUs/Tareas/FB_TransferirPale_SFC.TcPOU
FUNCTION_BLOCK FB_TransferirPale_SFC
VAR_INPUT
	
	//Tiempo
	Tcheck: TIME := T#1S;	

	// SFC-Flags
	SFCPause: BOOL;
	SFCReset: BOOL;
	
	//Indicadores de sincronizacion
	Ack: BOOL:= TRUE;
	Execute: BOOL;
	
	//Entradas
	Presencia_pale:BOOL;

	
END_VAR
VAR_OUTPUT
	//indicadores de sincronizacion
	Done: BOOL;
	Ready: BOOL;

	//Salidas
	Retenedor_pale_baja: BOOL;
	Activa_marcha_motor_cinta: BOOL;
	Separador_pale_sube: BOOL;
	
END_VAR
VAR
END_VAR

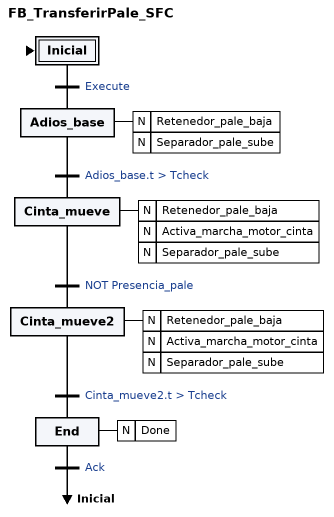
INITIAL_STEP Inicial:
END_STEP
TRANSITION FROM Inicial TO Adios_base
    := Execute;
END_TRANSITION
STEP Adios_base:
    Retenedor_pale_baja(N);
    Separador_pale_sube(N);
END_STEP
TRANSITION FROM Adios_base TO Cinta_mueve
    := Adios_base.t > Tcheck;
END_TRANSITION
STEP Cinta_mueve:
    Retenedor_pale_baja(N);
    Activa_marcha_motor_cinta(N);
    Separador_pale_sube(N);
END_STEP
TRANSITION FROM Cinta_mueve TO Cinta_mueve2
    := NOT Presencia_pale;
END_TRANSITION
STEP Cinta_mueve2:
    Retenedor_pale_baja(N);
    Activa_marcha_motor_cinta(N);
    Separador_pale_sube(N);
END_STEP
TRANSITION FROM Cinta_mueve2 TO End
    := Cinta_mueve2.t > Tcheck;
END_TRANSITION
STEP End:
    Done(N);
END_STEP
TRANSITION FROM End TO Inicial
    := Ack;
END_TRANSITION

END_FUNCTION_BLOCK

// ---- POUs/Tareas/FB_EstacionFinalizar_SFC.TcPOU
FUNCTION_BLOCK FB_EstacionFinalizar_SFC
VAR_INPUT

    // SFC-Flags
    SFCPause: BOOL;
    SFCReset: BOOL;

    // Indicadores de sincronizacion
    Ack: BOOL := TRUE;
    Execute: BOOL;

   //Entradas
    Horizontal_descargador_detras: BOOL;
	Vertical_descargador_arriba: BOOL;
	Presencia_pale: BOOL;
	
END_VAR
VAR_OUTPUT
    // Indicadores de sincronizacion
    Done: BOOL;
    Ready: BOOL;
	
	//Salidas
	Descargador_atras: BOOL;
	Activa_marcha_motor_cinta: BOOL;
END_VAR
VAR
	Tcinta: TIME := T#0.5S;
END_VAR

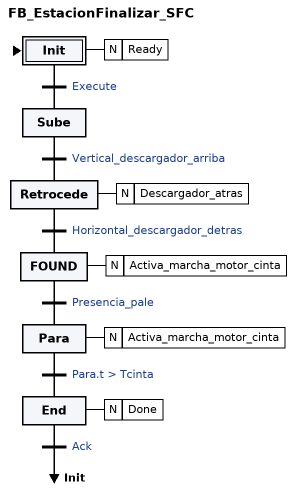
INITIAL_STEP Init:
    Ready(N);
END_STEP
TRANSITION FROM Init TO Sube
    := Execute;
END_TRANSITION
STEP Sube:
END_STEP
TRANSITION FROM Sube TO Retrocede
    := Vertical_descargador_arriba;
END_TRANSITION
STEP Retrocede:
    Descargador_atras(N);
END_STEP
TRANSITION FROM Retrocede TO FOUND
    := Horizontal_descargador_detras;
END_TRANSITION
STEP FOUND:
    Activa_marcha_motor_cinta(N);
END_STEP
TRANSITION FROM FOUND TO Para
    := Presencia_pale;
END_TRANSITION
STEP Para:
    Activa_marcha_motor_cinta(N);
END_STEP
TRANSITION FROM Para TO End
    := Para.t > Tcinta;
END_TRANSITION
STEP End:
    Done(N);
END_STEP
TRANSITION FROM End TO Init
    := Ack;
END_TRANSITION

END_FUNCTION_BLOCK

// ---- POUs/Tareas/FB_EstacionPreparar_SFC.TcPOU
FUNCTION_BLOCK FB_EstacionPreparar_SFC
VAR_INPUT

    // SFC-Flags
    SFCPause: BOOL;
    SFCReset: BOOL;

    // Indicadores de sincronizacion
    Ack: BOOL := TRUE;
    Execute: BOOL;

   //Entradas
    Horizontal_descargador_detras: BOOL;
	Vertical_descargador_arriba: BOOL;
	Presencia_pale: BOOL;
	
END_VAR
VAR_OUTPUT
    // Indicadores de sincronizacion
    Done: BOOL;
    Ready: BOOL;
	
	//Salidas
	Descargador_atras: BOOL;
	Activa_marcha_motor_cinta: BOOL;
END_VAR
VAR
	Tcinta: TIME := T#0.5S;
END_VAR

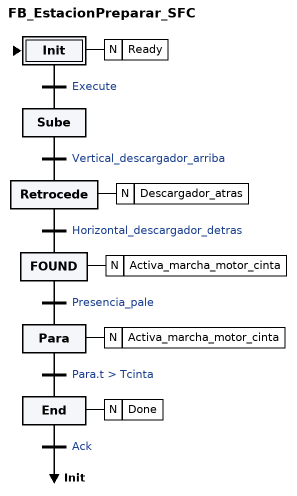
INITIAL_STEP Init:
    Ready(N);
END_STEP
TRANSITION FROM Init TO Sube
    := Execute;
END_TRANSITION
STEP Sube:
END_STEP
TRANSITION FROM Sube TO Retrocede
    := Vertical_descargador_arriba;
END_TRANSITION
STEP Retrocede:
    Descargador_atras(N);
END_STEP
TRANSITION FROM Retrocede TO FOUND
    := Horizontal_descargador_detras;
END_TRANSITION
STEP FOUND:
    Activa_marcha_motor_cinta(N);
END_STEP
TRANSITION FROM FOUND TO Para
    := Presencia_pale;
END_TRANSITION
STEP Para:
    Activa_marcha_motor_cinta(N);
END_STEP
TRANSITION FROM Para TO End
    := Para.t > Tcinta;
END_TRANSITION
STEP End:
    Done(N);
END_STEP
TRANSITION FROM End TO Init
    := Ack;
END_TRANSITION

END_FUNCTION_BLOCK

// ---- GlobalTextList.TcGTLO
TEXTLIST GlobalTextList
  939 = '%d'
  602 = '%s'
  833 = '+'
  832 = '-'
  402 = '.0'
  16 = '.1'
  415 = '.2'
  831 = '0'
  830 = '1'
  834 = '2'
  3 = '2023'
  827 = '3'
  39 = '4'
  583 = 'A'
  743 = 'Alto'
  739 = 'B'
  984 = 'Bajo'
  782 = 'C'
  941 = 'Cargador Cilindro'
  486 = 'Cargador Eyector'
  228 = 'CI'
  912 = 'Cinta Motor'
  423 = 'Cinta Retenedor'
  852 = 'Cinta Separador'
  951 = 'Conectada'
  122 = 'cp'
  419 = 'Código Palé'
  820 = 'D'
  1323 = 'Desconecta'
  469 = 'E'
  695 = 'Emergencia'
  87 = 'Entrada Palé'
  585 = 'Estructurado'
  902 = 'Extractor'
  896 = 'FMS-203'
  243 = 'GEMMA'
  489 = 'Grupo Hidráulico'
  222 = 'H'
  129 = 'Hidráulico'
  524 = 'Introductor'
  372 = 'ISA'
  531 = 'KM'
  927 = 'L. Alarma'
  664 = 'L. Marcha'
  537 = 'Manipulador'
  287 = 'Manipulador Cilindro'
  139 = 'Manipulador Eyector'
  923 = 'Manual'
  332 = 'Modo'
  544 = 'P. Marcha'
  15 = 'P. Parada'
  438 = 'PANEL'
  584 = 'PARÁMETROS'
  37 = 'Pausa'
  513 = 'Pendientes'
  284 = 'PLANTA'
  676 = 'pp'
  424 = 'PRENSADO HIDRÁULICO DEL RODAMIENTO'
  64 = 'Prensador'
  366 = 'Presostato'
  258 = 'Protector'
  171 = 'R'
  915 = 'Realizadas'
  328 = 'Reposo'
  621 = 'Reset'
  190 = 'Retenedor'
  248 = 'S'
  949 = 'Salida Palé'
  693 = 'Separador'
  333 = 'Solicitadas'
  390 = 'TAREA'
  569 = 'Transf. Palé'
  441 = 'V'
END_TEXTLIST

// ---- VISUs/Visualization.TcVIS
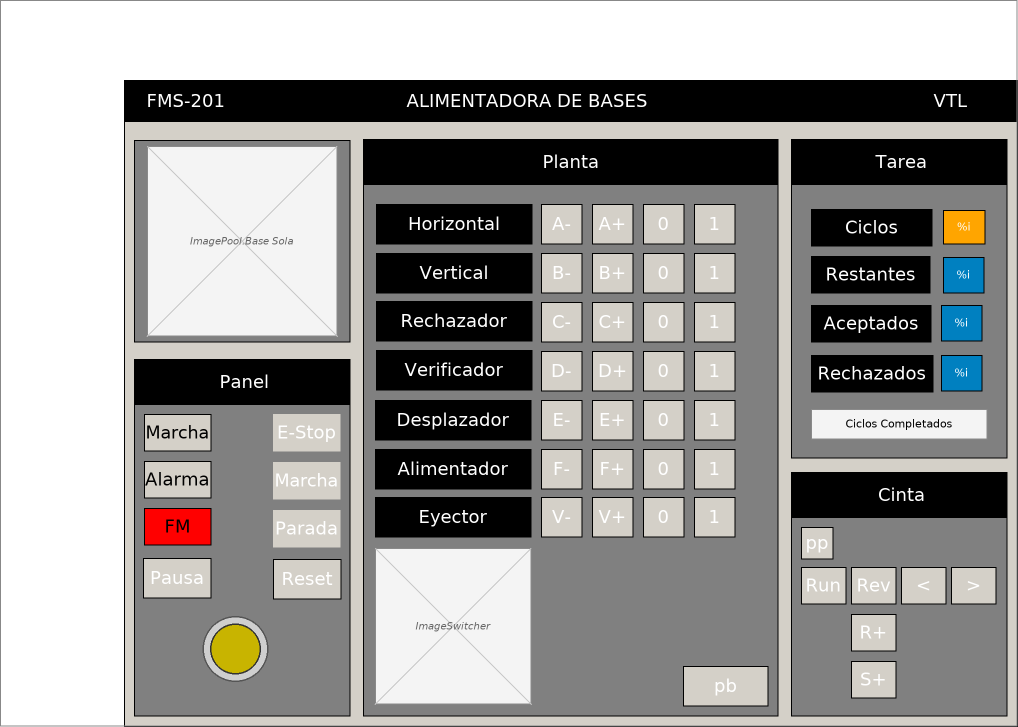
VISUALIZATION Visualization  // 1018x727
    Rectangle (124,121 894x606)
    Rectangle (791,184 216x274)
    Rectangle (363,184 415x532)
    Rectangle (363,139 415x45)
    Label (363,141 416x42), "Planta"
    Rectangle (791,139 216x45)
    Label (841,144 121x36), "Tarea"
    Progressbar (811,409 176x30), "Ciclos Completados", variable: MAIN.test_pieza.Aceptados
    RoundedRectangle (376,204 156x40), "Horizontal"
    Textfield (943,210 42x34), "%i", text variable: MAIN.Estacion.CiclosSolicitados
        OnMouseDown: write MAIN.Estacion.CiclosSolicitados via VisuDialogs.Numpad, min 1, max 10
    RoundedRectangle (811,209 121x37), "Ciclos"
    RoundedRectangle (811,256 119x37), "Restantes"
    RoundedRectangle (811,305 120x37), "Aceptados"
    RoundedRectangle (811,355 122x37), "Rechazados"
    Textfield (943,257 41x36), "%i", text variable: MAIN.Estacion.CiclosPendientes
    Textfield (941,305 41x36), "%i", text variable: MAIN.Estacion.CiclosAceptados
    Textfield (941,355 41x36), "%i", text variable: MAIN.Estacion.CiclosRechazados
    RoundedRectangle (592,253 41x40), "B+", colour toggle: MAIN.Estacion.Descargador_baja
        toggle MAIN.Estacion.Descargador_baja
    Rectangle (791,517 216x199)
    Rectangle (791,472 216x45)
    Label (841,477 121x36), "Cinta"
    Rectangle (134,140 216x202)
    Rectangle (134,404 216x312)
    Rectangle (134,359 216x45)
    Label (184,364 121x36), "Panel"
    Rectangle (124,80 894x41)
    Label (124,81 893x40), "FMS-201 ALIMENTADORA DE BASES VTL"
    RoundedRectangle (376,253 156x40), "Vertical"
    RoundedRectangle (592,204 41x40), "A+", colour toggle: MAIN.Estacion.Descargador_adelante
        tap MAIN.Estacion.Descargador_adelante
    RoundedRectangle (592,302 41x40), "C+", colour toggle: MAIN.Estacion.Rechazador_adelante
        tap MAIN.Estacion.Rechazador_adelante
    RoundedRectangle (592,351 41x40), "D+", colour toggle: MAIN.Estacion.Verificador_baja
        tap MAIN.Estacion.Verificador_baja
    RoundedRectangle (592,400 41x40), "E+", colour toggle: MAIN.Estacion.Desplazador_adelante
        tap MAIN.Estacion.Desplazador_adelante
    RoundedRectangle (592,449 41x40), "F+", colour toggle: MAIN.Estacion.Alimentador_adelante
        tap MAIN.Estacion.Alimentador_adelante
    RoundedRectangle (592,497 41x40), "V+", colour toggle: MAIN.Estacion.Eyector_succiona
        toggle MAIN.Estacion.Eyector_succiona
    RoundedRectangle (376,301 156x40), "Rechazador"
    RoundedRectangle (376,350 156x40), "Verificador"
    RoundedRectangle (375,400 156x40), "Desplazador"
    RoundedRectangle (375,449 156x40), "Alimentador"
    RoundedRectangle (375,497 156x40), "Eyector"
    RoundedRectangle (541,204 41x40), "A-", colour toggle: MAIN.Estacion.Descargador_atras
        tap MAIN.Estacion.Descargador_atras
    RoundedRectangle (643,204 41x40), "0", colour toggle: MAIN.Estacion.Horizontal_descargador_detras
    RoundedRectangle (694,204 41x40), "1", colour toggle: MAIN.Estacion.Horizontal_descargador_delante
    RoundedRectangle (643,253 41x40), "0", colour toggle: MAIN.Estacion.Vertical_descargador_arriba
        tap MAIN.Estacion.Vertical_descargador_arriba
    RoundedRectangle (694,253 41x40), "1", colour toggle: MAIN.Estacion.Vertical_descargador_abajo
        tap MAIN.Estacion.Vertical_descargador_abajo
    RoundedRectangle (643,302 41x40), "0"
    RoundedRectangle (643,351 41x40), "0", colour toggle: MAIN.Estacion.Verificador_arriba
        tap MAIN.Estacion.Verificador_arriba
    RoundedRectangle (643,400 41x40), "0", colour toggle: MAIN.Estacion.Desplazador_detras
        tap MAIN.Estacion.Desplazador_detras
    RoundedRectangle (643,449 41x40), "0", colour toggle: MAIN.Estacion.Alimentador_detras
        tap MAIN.Estacion.Alimentador_detras
    RoundedRectangle (643,497 41x40), "0"
    RoundedRectangle (694,302 41x40), "1"
    RoundedRectangle (694,351 41x40), "1", colour toggle: MAIN.Estacion.Verificador_abajo
        tap MAIN.Estacion.Verificador_abajo
    RoundedRectangle (694,400 41x40), "1"
    RoundedRectangle (694,449 41x40), "1", colour toggle: MAIN.Estacion.Alimentador_delante
        tap MAIN.Estacion.Alimentador_delante
    RoundedRectangle (694,497 41x40), "1", colour toggle: MAIN.Estacion.Vacio_obtenido_vacuostato_descargador
        tap MAIN.Estacion.Vacio_obtenido_vacuostato_descargador
    RoundedRectangle (541,253 41x40), "B-"
    RoundedRectangle (541,302 41x40), "C-"
    RoundedRectangle (541,351 41x40), "D-"
    RoundedRectangle (541,400 41x40), "E-"
    RoundedRectangle (541,449 41x40), "F-"
    RoundedRectangle (541,497 41x40), "V-"
    RoundedRectangle (683,666 85x40), "pb", colour toggle: MAIN.Estacion.Base_en_Alimentador
        tap MAIN.Estacion.Base_en_Alimentador
    RoundedRectangle (144,508 67x37), "FM", colour toggle: MAIN.Estacion.Lampara_falta_material
        tap MAIN.Estacion.Lampara_falta_material
    RoundedRectangle (801,527 32x32), "pp", colour toggle: MAIN.Estacion.Presencia_pale
        tap MAIN.Estacion.Presencia_pale
    RoundedRectangle (951,567 45x37), ">", colour toggle: MAIN.Estacion.Activa_marcha_motor_cinta
        tap MAIN.Estacion.Activa_marcha_motor_cinta
    RoundedRectangle (901,567 45x37), "<", colour toggle: MAIN.Estacion.Invierte_marcha_motor_cinta
        toggle MAIN.Estacion.Invierte_marcha_motor_cinta
    RoundedRectangle (801,567 45x37), "Run", colour toggle: MAIN.Estacion.Activa_marcha_motor_cinta
    RoundedRectangle (851,567 45x37), "Rev", colour toggle: MAIN.Estacion.Invierte_marcha_motor_cinta
    RoundedRectangle (851,614 45x37), "R+", colour toggle: MAIN.Estacion.Retenedor_pale_baja
        toggle MAIN.Estacion.Retenedor_pale_baja
    RoundedRectangle (851,661 45x37), "S+", colour toggle: MAIN.Estacion.Separador_pale_sube
        toggle MAIN.Estacion.Separador_pale_sube
    RoundedRectangle (273,414 67x37), "E-Stop", colour toggle: MAIN.Estacion.Pulsador_parada_emergencia
        tap MAIN.Estacion.Pulsador_parada_emergencia
    RoundedRectangle (273,462 67x37), "Marcha", colour toggle: MAIN.Estacion.Pulsador_marcha
        tap MAIN.Estacion.Pulsador_marcha
    RoundedRectangle (273,510 67x37), "Parada", colour toggle: MAIN.Estacion.Pulsador_parada_NC
        tap MAIN.Estacion.Pulsador_parada_NC
    RoundedRectangle (144,461 67x37), "Alarma", colour toggle: MAIN.Estacion.Lampara_alarma
        tap MAIN.Estacion.Lampara_alarma
    RoundedRectangle (144,414 67x37), "Marcha", colour toggle: MAIN.Estacion.Lampara_marcha
        tap MAIN.Estacion.Lampara_marcha
    Image (147,146 190x190), image: ImagePool.Base Sola
    Lamp1 (197,611 77x76), variable: MAIN.test_pieza.Lampara_falta_material, style: Lamp-Lamp1-Yellow
    ImageSwitcher (375,548 156x156), variable: MAIN.Estacion.pieza_ok, background image: ImagePool.Base OK, image: ImagePool.Base No OK, behaviour: TOGGLE
    RoundedRectangle (143,558 68x40), "Pausa", text variable: MAIN.Estacion.EstadoPausa, colour toggle: MAIN.Estacion.EstadoPausaMAIN.Estacion.EstadoPausa
        tap MAIN.Estacion.EstadoPausa
    RoundedRectangle (273,559 68x40), "Reset", text variable: MAIN.Estacion.EstadoReinicia, colour toggle: MAIN.Estacion.EstadoReinicia
        tap MAIN.Estacion.EstadoReinicia
END_VISUALIZATION
